FUNCTION_BLOCK PressureInput EXTENDS AnalogInput
VAR_INPUT
	Range: LREAL := 32767;
END_VAR
VAR_OUTPUT
END_VAR
VAR
	Aver: Average;
END_VAR
VAR PERSISTENT
END_VAR

SUPER^();

METHOD FB_init : BOOL
VAR_INPUT
	bInitRetains : BOOL; // if TRUE, the retain variables are initialized (warm start / cold start)
	bInCopyCode : BOOL;  // if TRUE, the instance afterwards gets moved into the copy code (online change)
END_VAR
IF bInitRetains THEN
	ProcessMin := 0;
	ProcessMax := 30000;
	MinValue := 0;
	MaxValue := 30000;
END_IF
END_METHOD

METHOD GetValue : LREAL
VAR_INPUT
END_VAR
Aver(NewSample := (SUPER^.GetValue() / 32767) * Range);
GetValue := Aver.Value;
END_METHOD

END_FUNCTION_BLOCK

(* stored: Version 1.1.0.1, ProductVersion 3.1.4024.4
   POU PressureInput: Id {f67aaebf-eb74-43fd-9634-7b59ef2b5baa}, SpecialFunc None
   Method FB_init: Id {ba164769-91c8-4910-878e-3bfbdd95965c}
   Method GetValue: Id {08f2c029-ba38-454f-9a1e-911b2aaa688f} *)
